{attribute 'qualified_only'}
{attribute 'strict'}
{attribute 'to_string'}
TYPE E_DataStatus :
(
    Ok,
    WcError,   // working counter reports invalid data
    Stale      // WC valid but the input toggle hasn't changed for the timeout window
) UDINT;
END_TYPE

(* stored: Version 1.1.0.1
   DUT E_DataStatus: Id {d8c2cf4e-e120-4f9f-8b5f-9f3edc2fd6a4} *)
